ABB RobotStudio station: Proyecto_manipuladores_G3.rsstn

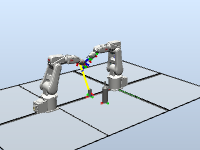
Station Proyecto_manipuladores (saved by RobotStudio format 3)
Controller Sistema8, task T_ROB1: task frame (RAPID world) sits at (1100, -1.84, 0) mm, rotated rx 0 ry 0 rz 180 deg in the station
Controller IRB_120_3kg_0.58m
  mechanical unit ROB_1: IRB120_3_58__01, 6 joints, base frame (0, 0, 0) mm
Controller Sistema8
  mechanical unit ROB_1: IRB120_3_58__01_3, 6 joints, base frame (0, 0, 0) mm
Layout (positions relative to the parent item):
  - IRB120_3_58__01 [mechanism, from Robots\IRB120_3_58_G_01.rslib] at (0, 0, 0) mm; joint values [0.0001, 0.0287, -0.0253, -0.0001, 0.5202, 0.0001] (rad or m)
  - Smart_Gripper_Servo_Fingers [mechanism, from Tools\ABB_Smart_Gripper_Servo_Fingers.rslib] at (372.35, 0.02, 592.85) mm, rotated rx 180 ry 60 rz 180 deg; joint values [0.025] (rad or m)
  - Botella_vino_objeto [part] at (0.08, -0.09, 0.03) mm, rotated rx 0 ry 0 rz 0.01 deg
  - Vaso [part] at (0, -0.1, -0.01) mm, rotated rx 0.01 ry 0 rz 0.01 deg
  - IRB120_3_58__01_3 [mechanism, from Robots\IRB120_3_58_G_01.rslib] at (1100, -1.84, 0) mm, rotated rx 0 ry 0 rz -180 deg; joint values [0, 0.3812, -0.2541, -0.0001, 0.3964, 0.0001] (rad or m)
  - Smart_Gripper_Servo_Fingers_2 [mechanism, from Tools\ABB_Smart_Gripper_Servo_Fingers.rslib] at (628.75, -1.86, 535.75) mm, rotated rx -180 ry 60 rz 0 deg; joint values [0.0221] (rad or m)
Attachment: Botella_vino is attached to Botella_vino_objeto
Attachment: Vasito is attached to Vaso
Attachment: Smart_Gripper_Servo_Fingers is attached to IRB120_3_58__01 / Link6
Attachment: Smart_Gripper_Servo_Fingers_2 is attached to IRB120_3_58__01_3 / Link6
EventTableEntry 1530: Group=, Trigger=Gripper 1531, Actions=[EventTableActionMechanicalPose 1532, EventTableActionAttach 1533], Comment=, ActivationMode=2, Cyclic=false
EventTableTriggerIO 1531: IOValue=[1], IRC5Controller=? -1, Operator=0, SignalSource=IRB_120_3kg_0.58m 521
EventTableActionMechanicalPose 1532: VirtualSignal=, Mechanism=Smart_Gripper_Servo_Fingers 1411, ToPoseName=CerradoVino, VirtualSignalValue=[1]
EventTableActionAttach 1533: AttachmentParent=Smart_Gripper_Servo_Fingers 1411, AttachmentChild=? -1, MountObject=false, Offset=[X=1, Y=0, Z=0, W=0, X=0, Y=1, Z=0, W=0, X=0, Y=0, Z=1, W=0, X=0, Y=0, Z=0, W=1], FlangeIndext=0, FindNearest=true
EventTableTriggerIO 1534: IOValue=[1], IRC5Controller=? -1, Operator=0, SignalSource=IRB_120_3kg_0.58m 521
EventTableTriggerIO 1535: IOValue=[1], IRC5Controller=? -1, Operator=0, SignalSource=IRB_120_3kg_0.58m 521
EventTableEntry 1536: Group=, Trigger=Gripper 1537, Actions=[EventTableActionMechanicalPose 1538, EventTableActionDetach 1539], Comment=, ActivationMode=2, Cyclic=false
EventTableTriggerIO 1537: IOValue=[0], IRC5Controller=? -1, Operator=0, SignalSource=IRB_120_3kg_0.58m 521
EventTableActionMechanicalPose 1538: VirtualSignal=, Mechanism=Smart_Gripper_Servo_Fingers 1411, ToPoseName=PoseAbierto, VirtualSignalValue=[1]
EventTableActionDetach 1539: AttachmentParent=Smart_Gripper_Servo_Fingers 1411, AttachmentChild=? -1
EventTableTriggerIO 1540: IOValue=[0], IRC5Controller=? -1, Operator=0, SignalSource=IRB_120_3kg_0.58m 521
EventTableTriggerIO 1541: IOValue=[0], IRC5Controller=? -1, Operator=0, SignalSource=IRB_120_3kg_0.58m 521
EventTableTriggerIO 1596: IOValue=[1], IRC5Controller=? -1, Operator=0, SignalSource=IRB_120_3kg_0.58m 521
EventTableTriggerIO 1597: IOValue=[1], IRC5Controller=? -1, Operator=0, SignalSource=IRB_120_3kg_0.58m 521
EventTableTriggerIO 1598: IOValue=[1], IRC5Controller=? -1, Operator=0, SignalSource=IRB_120_3kg_0.58m 521
EventTableTriggerIO 1599: IOValue=[0], IRC5Controller=? -1, Operator=0, SignalSource=IRB_120_3kg_0.58m 521
EventTableTriggerIO 1600: IOValue=[0], IRC5Controller=? -1, Operator=0, SignalSource=IRB_120_3kg_0.58m 521
EventTableTriggerIO 1601: IOValue=[0], IRC5Controller=? -1, Operator=0, SignalSource=IRB_120_3kg_0.58m 521
EventTableTriggerIO 1602: IOValue=[1], IRC5Controller=? -1, Operator=0, SignalSource=IRB_120_3kg_0.58m 521
EventTableTriggerIO 1603: IOValue=[0], IRC5Controller=? -1, Operator=0, SignalSource=IRB_120_3kg_0.58m 521
EventTableTriggerIO 1604: IOValue=[1], IRC5Controller=? -1, Operator=0, SignalSource=IRB_120_3kg_0.58m 521
EventTableTriggerIO 1605: IOValue=[1], IRC5Controller=? -1, Operator=0, SignalSource=IRB_120_3kg_0.58m 521
EventTableTriggerIO 1606: IOValue=[1], IRC5Controller=? -1, Operator=0, SignalSource=IRB_120_3kg_0.58m 521
EventTableTriggerIO 1607: IOValue=[1], IRC5Controller=? -1, Operator=0, SignalSource=IRB_120_3kg_0.58m 521
EventTableTriggerIO 1608: IOValue=[0], IRC5Controller=? -1, Operator=0, SignalSource=IRB_120_3kg_0.58m 521
EventTableTriggerIO 1609: IOValue=[0], IRC5Controller=? -1, Operator=0, SignalSource=IRB_120_3kg_0.58m 521
EventTableTriggerIO 1610: IOValue=[0], IRC5Controller=? -1, Operator=0, SignalSource=IRB_120_3kg_0.58m 521
EventTableTriggerIO 1611: IOValue=[0], IRC5Controller=? -1, Operator=0, SignalSource=IRB_120_3kg_0.58m 521
EventTableTriggerIO 1646: IOValue=[1], IRC5Controller=? -1, Operator=0, SignalSource=IRB_120_3kg_0.58m 521
EventTableTriggerIO 1647: IOValue=[1], IRC5Controller=? -1, Operator=0, SignalSource=IRB_120_3kg_0.58m 521
EventTableTriggerIO 1648: IOValue=[0], IRC5Controller=? -1, Operator=0, SignalSource=IRB_120_3kg_0.58m 521
EventTableTriggerIO 1649: IOValue=[0], IRC5Controller=? -1, Operator=0, SignalSource=IRB_120_3kg_0.58m 521
EventTableTriggerIO 1667: IOValue=[1], IRC5Controller=? -1, Operator=0, SignalSource=IRB_120_3kg_0.58m 521
EventTableTriggerIO 1668: IOValue=[1], IRC5Controller=? -1, Operator=0, SignalSource=IRB_120_3kg_0.58m 521
EventTableTriggerIO 1669: IOValue=[1], IRC5Controller=? -1, Operator=0, SignalSource=IRB_120_3kg_0.58m 521
EventTableTriggerIO 1670: IOValue=[1], IRC5Controller=? -1, Operator=0, SignalSource=IRB_120_3kg_0.58m 521
EventTableTriggerIO 1671: IOValue=[1], IRC5Controller=? -1, Operator=0, SignalSource=IRB_120_3kg_0.58m 521
EventTableTriggerIO 1672: IOValue=[1], IRC5Controller=? -1, Operator=0, SignalSource=IRB_120_3kg_0.58m 521
EventTableTriggerIO 1673: IOValue=[1], IRC5Controller=? -1, Operator=0, SignalSource=IRB_120_3kg_0.58m 521
EventTableTriggerIO 1674: IOValue=[1], IRC5Controller=? -1, Operator=0, SignalSource=IRB_120_3kg_0.58m 521
EventTableTriggerIO 1675: IOValue=[1], IRC5Controller=? -1, Operator=0, SignalSource=IRB_120_3kg_0.58m 521
EventTableTriggerIO 1676: IOValue=[0], IRC5Controller=? -1, Operator=0, SignalSource=IRB_120_3kg_0.58m 521
EventTableTriggerIO 1677: IOValue=[0], IRC5Controller=? -1, Operator=0, SignalSource=IRB_120_3kg_0.58m 521
EventTableTriggerIO 1678: IOValue=[0], IRC5Controller=? -1, Operator=0, SignalSource=IRB_120_3kg_0.58m 521
EventTableTriggerIO 1679: IOValue=[0], IRC5Controller=? -1, Operator=0, SignalSource=IRB_120_3kg_0.58m 521
EventTableTriggerIO 1680: IOValue=[0], IRC5Controller=? -1, Operator=0, SignalSource=IRB_120_3kg_0.58m 521
EventTableTriggerIO 1681: IOValue=[0], IRC5Controller=? -1, Operator=0, SignalSource=IRB_120_3kg_0.58m 521
EventTableTriggerIO 1682: IOValue=[0], IRC5Controller=? -1, Operator=0, SignalSource=IRB_120_3kg_0.58m 521
EventTableTriggerIO 1683: IOValue=[0], IRC5Controller=? -1, Operator=0, SignalSource=IRB_120_3kg_0.58m 521
EventTableTriggerIO 1684: IOValue=[0], IRC5Controller=? -1, Operator=0, SignalSource=IRB_120_3kg_0.58m 521
EventTableTriggerIO 2365: IOValue=[1], IRC5Controller=? -1, Operator=0, SignalSource=IRB_120_3kg_0.58m 521
EventTableTriggerIO 2366: IOValue=[1], IRC5Controller=? -1, Operator=0, SignalSource=IRB_120_3kg_0.58m 521
EventTableTriggerIO 2367: IOValue=[1], IRC5Controller=? -1, Operator=0, SignalSource=IRB_120_3kg_0.58m 521
EventTableTriggerIO 2368: IOValue=[1], IRC5Controller=? -1, Operator=0, SignalSource=IRB_120_3kg_0.58m 521
EventTableTriggerIO 2369: IOValue=[1], IRC5Controller=? -1, Operator=0, SignalSource=IRB_120_3kg_0.58m 521
EventTableTriggerIO 2370: IOValue=[1], IRC5Controller=? -1, Operator=0, SignalSource=IRB_120_3kg_0.58m 521
EventTableTriggerIO 2371: IOValue=[1], IRC5Controller=? -1, Operator=0, SignalSource=IRB_120_3kg_0.58m 521
EventTableTriggerIO 2372: IOValue=[1], IRC5Controller=? -1, Operator=0, SignalSource=IRB_120_3kg_0.58m 521
EventTableTriggerIO 2373: IOValue=[1], IRC5Controller=? -1, Operator=0, SignalSource=IRB_120_3kg_0.58m 521
EventTableTriggerIO 2374: IOValue=[0], IRC5Controller=? -1, Operator=0, SignalSource=IRB_120_3kg_0.58m 521
EventTableTriggerIO 2375: IOValue=[0], IRC5Controller=? -1, Operator=0, SignalSource=IRB_120_3kg_0.58m 521
EventTableTriggerIO 2376: IOValue=[0], IRC5Controller=? -1, Operator=0, SignalSource=IRB_120_3kg_0.58m 521
EventTableTriggerIO 2377: IOValue=[0], IRC5Controller=? -1, Operator=0, SignalSource=IRB_120_3kg_0.58m 521
EventTableTriggerIO 2378: IOValue=[0], IRC5Controller=? -1, Operator=0, SignalSource=IRB_120_3kg_0.58m 521
EventTableTriggerIO 2379: IOValue=[0], IRC5Controller=? -1, Operator=0, SignalSource=IRB_120_3kg_0.58m 521
EventTableTriggerIO 2380: IOValue=[0], IRC5Controller=? -1, Operator=0, SignalSource=IRB_120_3kg_0.58m 521
EventTableTriggerIO 2381: IOValue=[0], IRC5Controller=? -1, Operator=0, SignalSource=IRB_120_3kg_0.58m 521
EventTableTriggerIO 2382: IOValue=[0], IRC5Controller=? -1, Operator=0, SignalSource=IRB_120_3kg_0.58m 521
EventTableTriggerIO 2468: IOValue=[1], IRC5Controller=? -1, Operator=0, SignalSource=Sistema8 2502
EventTableTriggerIO 2469: IOValue=[0], IRC5Controller=? -1, Operator=0, SignalSource=Sistema8 2502
EventTableTriggerIO 2470: IOValue=[1], IRC5Controller=? -1, Operator=0, SignalSource=IRB_120_3kg_0.58m 521
EventTableTriggerIO 2471: IOValue=[1], IRC5Controller=? -1, Operator=0, SignalSource=Sistema8 2502
EventTableTriggerIO 2472: IOValue=[0], IRC5Controller=? -1, Operator=0, SignalSource=Sistema8 2502
EventTableTriggerIO 2473: IOValue=[1], IRC5Controller=? -1, Operator=0, SignalSource=IRB_120_3kg_0.58m 521
EventTableTriggerIO 2474: IOValue=[1], IRC5Controller=? -1, Operator=0, SignalSource=Sistema8 2502
EventTableTriggerIO 2475: IOValue=[0], IRC5Controller=? -1, Operator=0, SignalSource=Sistema8 2502
EventTableTriggerIO 2476: IOValue=[1], IRC5Controller=? -1, Operator=0, SignalSource=IRB_120_3kg_0.58m 521
EventTableTriggerIO 2477: IOValue=[1], IRC5Controller=? -1, Operator=0, SignalSource=Sistema8 2502
EventTableTriggerIO 2478: IOValue=[0], IRC5Controller=? -1, Operator=0, SignalSource=Sistema8 2502
EventTableTriggerIO 2479: IOValue=[1], IRC5Controller=? -1, Operator=0, SignalSource=IRB_120_3kg_0.58m 521
EventTableTriggerIO 2480: IOValue=[1], IRC5Controller=? -1, Operator=0, SignalSource=Sistema8 2502
EventTableTriggerIO 2481: IOValue=[0], IRC5Controller=? -1, Operator=0, SignalSource=Sistema8 2502
EventTableTriggerIO 2482: IOValue=[1], IRC5Controller=? -1, Operator=0, SignalSource=IRB_120_3kg_0.58m 521
EventTableTriggerIO 2483: IOValue=[1], IRC5Controller=? -1, Operator=0, SignalSource=Sistema8 2502
EventTableTriggerIO 2484: IOValue=[0], IRC5Controller=? -1, Operator=0, SignalSource=Sistema8 2502
EventTableTriggerIO 2485: IOValue=[1], IRC5Controller=? -1, Operator=0, SignalSource=IRB_120_3kg_0.58m 521
EventTableTriggerIO 2486: IOValue=[1], IRC5Controller=? -1, Operator=0, SignalSource=Sistema8 2502
EventTableTriggerIO 2487: IOValue=[0], IRC5Controller=? -1, Operator=0, SignalSource=Sistema8 2502
EventTableTriggerIO 2488: IOValue=[0], IRC5Controller=? -1, Operator=0, SignalSource=IRB_120_3kg_0.58m 521
EventTableTriggerIO 2489: IOValue=[0], IRC5Controller=? -1, Operator=0, SignalSource=IRB_120_3kg_0.58m 521
EventTableTriggerIO 2490: IOValue=[0], IRC5Controller=? -1, Operator=0, SignalSource=IRB_120_3kg_0.58m 521
EventTableTriggerIO 2491: IOValue=[0], IRC5Controller=? -1, Operator=0, SignalSource=IRB_120_3kg_0.58m 521
EventTableTriggerIO 2492: IOValue=[0], IRC5Controller=? -1, Operator=0, SignalSource=IRB_120_3kg_0.58m 521
EventTableTriggerIO 2493: IOValue=[0], IRC5Controller=? -1, Operator=0, SignalSource=IRB_120_3kg_0.58m 521
EventTableEntry 2494: Group=, Trigger=Gripper2 2468, Actions=[EventTableActionMechanicalPose 2495, EventTableActionAttach 2496], Comment=, ActivationMode=2, Cyclic=false
EventTableActionMechanicalPose 2495: VirtualSignal=, Mechanism=Smart_Gripper_Servo_Fingers_2 3134, ToPoseName=PoseAbre, VirtualSignalValue=[1]
EventTableActionAttach 2496: AttachmentParent=Smart_Gripper_Servo_Fingers_2 3134, AttachmentChild=? -1, MountObject=false, Offset=[X=1, Y=0, Z=0, W=0, X=0, Y=1, Z=0, W=0, X=0, Y=0, Z=1, W=0, X=0, Y=0, Z=0, W=1], FlangeIndext=0, FindNearest=true
EventTableEntry 2497: Group=, Trigger=Gripper2 2469, Actions=[EventTableActionMechanicalPose 3306, EventTableActionDetach 3307], Comment=, ActivationMode=2, Cyclic=false
EventTableTriggerIO 3106: IOValue=[1], IRC5Controller=? -1, Operator=0, SignalSource=IRB_120_3kg_0.58m 521
EventTableTriggerIO 3107: IOValue=[1], IRC5Controller=? -1, Operator=0, SignalSource=Sistema8 2502
EventTableTriggerIO 3108: IOValue=[0], IRC5Controller=? -1, Operator=0, SignalSource=Sistema8 2502
EventTableTriggerIO 3109: IOValue=[1], IRC5Controller=? -1, Operator=0, SignalSource=IRB_120_3kg_0.58m 521
EventTableTriggerIO 3110: IOValue=[1], IRC5Controller=? -1, Operator=0, SignalSource=Sistema8 2502
EventTableTriggerIO 3111: IOValue=[0], IRC5Controller=? -1, Operator=0, SignalSource=Sistema8 2502
EventTableTriggerIO 3112: IOValue=[1], IRC5Controller=? -1, Operator=0, SignalSource=IRB_120_3kg_0.58m 521
EventTableTriggerIO 3113: IOValue=[1], IRC5Controller=? -1, Operator=0, SignalSource=Sistema8 2502
EventTableTriggerIO 3114: IOValue=[0], IRC5Controller=? -1, Operator=0, SignalSource=Sistema8 2502
EventTableTriggerIO 3115: IOValue=[1], IRC5Controller=? -1, Operator=0, SignalSource=IRB_120_3kg_0.58m 521
EventTableTriggerIO 3116: IOValue=[1], IRC5Controller=? -1, Operator=0, SignalSource=Sistema8 2502
EventTableTriggerIO 3117: IOValue=[0], IRC5Controller=? -1, Operator=0, SignalSource=Sistema8 2502
EventTableTriggerIO 3118: IOValue=[1], IRC5Controller=? -1, Operator=0, SignalSource=IRB_120_3kg_0.58m 521
EventTableTriggerIO 3119: IOValue=[1], IRC5Controller=? -1, Operator=0, SignalSource=Sistema8 2502
EventTableTriggerIO 3120: IOValue=[0], IRC5Controller=? -1, Operator=0, SignalSource=Sistema8 2502
EventTableTriggerIO 3121: IOValue=[1], IRC5Controller=? -1, Operator=0, SignalSource=IRB_120_3kg_0.58m 521
EventTableTriggerIO 3122: IOValue=[1], IRC5Controller=? -1, Operator=0, SignalSource=Sistema8 2502
EventTableTriggerIO 3123: IOValue=[0], IRC5Controller=? -1, Operator=0, SignalSource=Sistema8 2502
EventTableTriggerIO 3124: IOValue=[0], IRC5Controller=? -1, Operator=0, SignalSource=IRB_120_3kg_0.58m 521
EventTableTriggerIO 3125: IOValue=[0], IRC5Controller=? -1, Operator=0, SignalSource=IRB_120_3kg_0.58m 521
EventTableTriggerIO 3126: IOValue=[0], IRC5Controller=? -1, Operator=0, SignalSource=IRB_120_3kg_0.58m 521
EventTableTriggerIO 3127: IOValue=[0], IRC5Controller=? -1, Operator=0, SignalSource=IRB_120_3kg_0.58m 521
EventTableTriggerIO 3128: IOValue=[0], IRC5Controller=? -1, Operator=0, SignalSource=IRB_120_3kg_0.58m 521
EventTableTriggerIO 3129: IOValue=[0], IRC5Controller=? -1, Operator=0, SignalSource=IRB_120_3kg_0.58m 521
EventTableTriggerIO 3142: IOValue=[1], IRC5Controller=? -1, Operator=0, SignalSource=IRB_120_3kg_0.58m 521
EventTableTriggerIO 3143: IOValue=[1], IRC5Controller=? -1, Operator=0, SignalSource=Sistema8 2502
EventTableTriggerIO 3144: IOValue=[0], IRC5Controller=? -1, Operator=0, SignalSource=Sistema8 2502
EventTableTriggerIO 3145: IOValue=[1], IRC5Controller=? -1, Operator=0, SignalSource=IRB_120_3kg_0.58m 521
EventTableTriggerIO 3146: IOValue=[1], IRC5Controller=? -1, Operator=0, SignalSource=Sistema8 2502
EventTableTriggerIO 3147: IOValue=[0], IRC5Controller=? -1, Operator=0, SignalSource=Sistema8 2502
EventTableTriggerIO 3148: IOValue=[1], IRC5Controller=? -1, Operator=0, SignalSource=IRB_120_3kg_0.58m 521
EventTableTriggerIO 3149: IOValue=[1], IRC5Controller=? -1, Operator=0, SignalSource=Sistema8 2502
EventTableTriggerIO 3150: IOValue=[0], IRC5Controller=? -1, Operator=0, SignalSource=Sistema8 2502
EventTableTriggerIO 3151: IOValue=[1], IRC5Controller=? -1, Operator=0, SignalSource=IRB_120_3kg_0.58m 521
EventTableTriggerIO 3152: IOValue=[1], IRC5Controller=? -1, Operator=0, SignalSource=Sistema8 2502
EventTableTriggerIO 3153: IOValue=[0], IRC5Controller=? -1, Operator=0, SignalSource=Sistema8 2502
EventTableTriggerIO 3154: IOValue=[1], IRC5Controller=? -1, Operator=0, SignalSource=IRB_120_3kg_0.58m 521
EventTableTriggerIO 3155: IOValue=[1], IRC5Controller=? -1, Operator=0, SignalSource=Sistema8 2502
EventTableTriggerIO 3156: IOValue=[0], IRC5Controller=? -1, Operator=0, SignalSource=Sistema8 2502
EventTableTriggerIO 3157: IOValue=[1], IRC5Controller=? -1, Operator=0, SignalSource=IRB_120_3kg_0.58m 521
EventTableTriggerIO 3158: IOValue=[1], IRC5Controller=? -1, Operator=0, SignalSource=Sistema8 2502
EventTableTriggerIO 3159: IOValue=[0], IRC5Controller=? -1, Operator=0, SignalSource=Sistema8 2502
EventTableTriggerIO 3160: IOValue=[1], IRC5Controller=? -1, Operator=0, SignalSource=IRB_120_3kg_0.58m 521
EventTableTriggerIO 3161: IOValue=[1], IRC5Controller=? -1, Operator=0, SignalSource=Sistema8 2502
EventTableTriggerIO 3162: IOValue=[0], IRC5Controller=? -1, Operator=0, SignalSource=Sistema8 2502
EventTableTriggerIO 3163: IOValue=[1], IRC5Controller=? -1, Operator=0, SignalSource=IRB_120_3kg_0.58m 521
EventTableTriggerIO 3164: IOValue=[1], IRC5Controller=? -1, Operator=0, SignalSource=Sistema8 2502
EventTableTriggerIO 3165: IOValue=[0], IRC5Controller=? -1, Operator=0, SignalSource=Sistema8 2502
EventTableTriggerIO 3166: IOValue=[1], IRC5Controller=? -1, Operator=0, SignalSource=IRB_120_3kg_0.58m 521
EventTableTriggerIO 3167: IOValue=[1], IRC5Controller=? -1, Operator=0, SignalSource=Sistema8 2502
EventTableTriggerIO 3168: IOValue=[0], IRC5Controller=? -1, Operator=0, SignalSource=Sistema8 2502
EventTableTriggerIO 3169: IOValue=[1], IRC5Controller=? -1, Operator=0, SignalSource=IRB_120_3kg_0.58m 521
EventTableTriggerIO 3170: IOValue=[1], IRC5Controller=? -1, Operator=0, SignalSource=Sistema8 2502
EventTableTriggerIO 3171: IOValue=[0], IRC5Controller=? -1, Operator=0, SignalSource=Sistema8 2502
EventTableTriggerIO 3172: IOValue=[1], IRC5Controller=? -1, Operator=0, SignalSource=IRB_120_3kg_0.58m 521
EventTableTriggerIO 3173: IOValue=[1], IRC5Controller=? -1, Operator=0, SignalSource=Sistema8 2502
EventTableTriggerIO 3174: IOValue=[0], IRC5Controller=? -1, Operator=0, SignalSource=Sistema8 2502
EventTableTriggerIO 3175: IOValue=[1], IRC5Controller=? -1, Operator=0, SignalSource=IRB_120_3kg_0.58m 521
EventTableTriggerIO 3176: IOValue=[1], IRC5Controller=? -1, Operator=0, SignalSource=Sistema8 2502
EventTableTriggerIO 3177: IOValue=[0], IRC5Controller=? -1, Operator=0, SignalSource=Sistema8 2502
EventTableTriggerIO 3178: IOValue=[1], IRC5Controller=? -1, Operator=0, SignalSource=IRB_120_3kg_0.58m 521
EventTableTriggerIO 3179: IOValue=[1], IRC5Controller=? -1, Operator=0, SignalSource=Sistema8 2502
EventTableTriggerIO 3180: IOValue=[0], IRC5Controller=? -1, Operator=0, SignalSource=Sistema8 2502
EventTableTriggerIO 3181: IOValue=[1], IRC5Controller=? -1, Operator=0, SignalSource=IRB_120_3kg_0.58m 521
EventTableTriggerIO 3182: IOValue=[1], IRC5Controller=? -1, Operator=0, SignalSource=Sistema8 2502
EventTableTriggerIO 3183: IOValue=[0], IRC5Controller=? -1, Operator=0, SignalSource=Sistema8 2502
EventTableTriggerIO 3184: IOValue=[1], IRC5Controller=? -1, Operator=0, SignalSource=IRB_120_3kg_0.58m 521
EventTableTriggerIO 3185: IOValue=[1], IRC5Controller=? -1, Operator=0, SignalSource=Sistema8 2502
EventTableTriggerIO 3186: IOValue=[0], IRC5Controller=? -1, Operator=0, SignalSource=Sistema8 2502
EventTableTriggerIO 3187: IOValue=[1], IRC5Controller=? -1, Operator=0, SignalSource=IRB_120_3kg_0.58m 521
EventTableTriggerIO 3188: IOValue=[1], IRC5Controller=? -1, Operator=0, SignalSource=Sistema8 2502
EventTableTriggerIO 3189: IOValue=[0], IRC5Controller=? -1, Operator=0, SignalSource=Sistema8 2502
EventTableTriggerIO 3190: IOValue=[1], IRC5Controller=? -1, Operator=0, SignalSource=IRB_120_3kg_0.58m 521
EventTableTriggerIO 3191: IOValue=[1], IRC5Controller=? -1, Operator=0, SignalSource=Sistema8 2502
EventTableTriggerIO 3192: IOValue=[0], IRC5Controller=? -1, Operator=0, SignalSource=Sistema8 2502
EventTableTriggerIO 3193: IOValue=[1], IRC5Controller=? -1, Operator=0, SignalSource=IRB_120_3kg_0.58m 521
EventTableTriggerIO 3194: IOValue=[1], IRC5Controller=? -1, Operator=0, SignalSource=Sistema8 2502
EventTableTriggerIO 3195: IOValue=[0], IRC5Controller=? -1, Operator=0, SignalSource=Sistema8 2502
EventTableTriggerIO 3196: IOValue=[1], IRC5Controller=? -1, Operator=0, SignalSource=IRB_120_3kg_0.58m 521
EventTableTriggerIO 3197: IOValue=[1], IRC5Controller=? -1, Operator=0, SignalSource=Sistema8 2502
EventTableTriggerIO 3198: IOValue=[0], IRC5Controller=? -1, Operator=0, SignalSource=Sistema8 2502
EventTableTriggerIO 3199: IOValue=[1], IRC5Controller=? -1, Operator=0, SignalSource=IRB_120_3kg_0.58m 521
EventTableTriggerIO 3200: IOValue=[1], IRC5Controller=? -1, Operator=0, SignalSource=Sistema8 2502
EventTableTriggerIO 3201: IOValue=[0], IRC5Controller=? -1, Operator=0, SignalSource=Sistema8 2502
EventTableTriggerIO 3202: IOValue=[1], IRC5Controller=? -1, Operator=0, SignalSource=IRB_120_3kg_0.58m 521
EventTableTriggerIO 3203: IOValue=[1], IRC5Controller=? -1, Operator=0, SignalSource=Sistema8 2502
EventTableTriggerIO 3204: IOValue=[0], IRC5Controller=? -1, Operator=0, SignalSource=Sistema8 2502
EventTableTriggerIO 3205: IOValue=[1], IRC5Controller=? -1, Operator=0, SignalSource=IRB_120_3kg_0.58m 521
EventTableTriggerIO 3206: IOValue=[1], IRC5Controller=? -1, Operator=0, SignalSource=Sistema8 2502
EventTableTriggerIO 3207: IOValue=[0], IRC5Controller=? -1, Operator=0, SignalSource=Sistema8 2502
EventTableTriggerIO 3208: IOValue=[1], IRC5Controller=? -1, Operator=0, SignalSource=IRB_120_3kg_0.58m 521
EventTableTriggerIO 3209: IOValue=[1], IRC5Controller=? -1, Operator=0, SignalSource=Sistema8 2502
EventTableTriggerIO 3210: IOValue=[0], IRC5Controller=? -1, Operator=0, SignalSource=Sistema8 2502
EventTableTriggerIO 3211: IOValue=[1], IRC5Controller=? -1, Operator=0, SignalSource=IRB_120_3kg_0.58m 521
EventTableTriggerIO 3212: IOValue=[1], IRC5Controller=? -1, Operator=0, SignalSource=Sistema8 2502
EventTableTriggerIO 3213: IOValue=[0], IRC5Controller=? -1, Operator=0, SignalSource=Sistema8 2502
EventTableTriggerIO 3214: IOValue=[1], IRC5Controller=? -1, Operator=0, SignalSource=IRB_120_3kg_0.58m 521
EventTableTriggerIO 3215: IOValue=[1], IRC5Controller=? -1, Operator=0, SignalSource=Sistema8 2502
EventTableTriggerIO 3216: IOValue=[0], IRC5Controller=? -1, Operator=0, SignalSource=Sistema8 2502
EventTableTriggerIO 3217: IOValue=[1], IRC5Controller=? -1, Operator=0, SignalSource=IRB_120_3kg_0.58m 521
EventTableTriggerIO 3218: IOValue=[1], IRC5Controller=? -1, Operator=0, SignalSource=Sistema8 2502
EventTableTriggerIO 3219: IOValue=[0], IRC5Controller=? -1, Operator=0, SignalSource=Sistema8 2502
EventTableTriggerIO 3220: IOValue=[1], IRC5Controller=? -1, Operator=0, SignalSource=IRB_120_3kg_0.58m 521
EventTableTriggerIO 3221: IOValue=[1], IRC5Controller=? -1, Operator=0, SignalSource=Sistema8 2502
EventTableTriggerIO 3222: IOValue=[0], IRC5Controller=? -1, Operator=0, SignalSource=Sistema8 2502
EventTableTriggerIO 3223: IOValue=[1], IRC5Controller=? -1, Operator=0, SignalSource=IRB_120_3kg_0.58m 521
EventTableTriggerIO 3224: IOValue=[1], IRC5Controller=? -1, Operator=0, SignalSource=Sistema8 2502
EventTableTriggerIO 3225: IOValue=[0], IRC5Controller=? -1, Operator=0, SignalSource=Sistema8 2502
EventTableTriggerIO 3226: IOValue=[1], IRC5Controller=? -1, Operator=0, SignalSource=IRB_120_3kg_0.58m 521
EventTableTriggerIO 3227: IOValue=[1], IRC5Controller=? -1, Operator=0, SignalSource=Sistema8 2502
EventTableTriggerIO 3228: IOValue=[0], IRC5Controller=? -1, Operator=0, SignalSource=Sistema8 2502
EventTableTriggerIO 3229: IOValue=[1], IRC5Controller=? -1, Operator=0, SignalSource=IRB_120_3kg_0.58m 521
EventTableTriggerIO 3230: IOValue=[1], IRC5Controller=? -1, Operator=0, SignalSource=Sistema8 2502
EventTableTriggerIO 3231: IOValue=[0], IRC5Controller=? -1, Operator=0, SignalSource=Sistema8 2502
EventTableTriggerIO 3232: IOValue=[1], IRC5Controller=? -1, Operator=0, SignalSource=IRB_120_3kg_0.58m 521
EventTableTriggerIO 3233: IOValue=[1], IRC5Controller=? -1, Operator=0, SignalSource=Sistema8 2502
EventTableTriggerIO 3234: IOValue=[0], IRC5Controller=? -1, Operator=0, SignalSource=Sistema8 2502
EventTableTriggerIO 3235: IOValue=[1], IRC5Controller=? -1, Operator=0, SignalSource=IRB_120_3kg_0.58m 521
EventTableTriggerIO 3236: IOValue=[1], IRC5Controller=? -1, Operator=0, SignalSource=Sistema8 2502
EventTableTriggerIO 3237: IOValue=[0], IRC5Controller=? -1, Operator=0, SignalSource=Sistema8 2502
EventTableTriggerIO 3238: IOValue=[1], IRC5Controller=? -1, Operator=0, SignalSource=IRB_120_3kg_0.58m 521
EventTableTriggerIO 3239: IOValue=[1], IRC5Controller=? -1, Operator=0, SignalSource=Sistema8 2502
EventTableTriggerIO 3240: IOValue=[0], IRC5Controller=? -1, Operator=0, SignalSource=Sistema8 2502
EventTableTriggerIO 3241: IOValue=[1], IRC5Controller=? -1, Operator=0, SignalSource=IRB_120_3kg_0.58m 521
EventTableTriggerIO 3242: IOValue=[1], IRC5Controller=? -1, Operator=0, SignalSource=Sistema8 2502
EventTableTriggerIO 3243: IOValue=[0], IRC5Controller=? -1, Operator=0, SignalSource=Sistema8 2502
EventTableTriggerIO 3244: IOValue=[1], IRC5Controller=? -1, Operator=0, SignalSource=IRB_120_3kg_0.58m 521
EventTableTriggerIO 3245: IOValue=[1], IRC5Controller=? -1, Operator=0, SignalSource=Sistema8 2502
EventTableTriggerIO 3246: IOValue=[0], IRC5Controller=? -1, Operator=0, SignalSource=Sistema8 2502
EventTableTriggerIO 3247: IOValue=[1], IRC5Controller=? -1, Operator=0, SignalSource=IRB_120_3kg_0.58m 521
EventTableTriggerIO 3248: IOValue=[1], IRC5Controller=? -1, Operator=0, SignalSource=Sistema8 2502
EventTableTriggerIO 3249: IOValue=[0], IRC5Controller=? -1, Operator=0, SignalSource=Sistema8 2502
EventTableTriggerIO 3250: IOValue=[1], IRC5Controller=? -1, Operator=0, SignalSource=IRB_120_3kg_0.58m 521
EventTableTriggerIO 3251: IOValue=[1], IRC5Controller=? -1, Operator=0, SignalSource=Sistema8 2502
EventTableTriggerIO 3252: IOValue=[0], IRC5Controller=? -1, Operator=0, SignalSource=Sistema8 2502
EventTableTriggerIO 3253: IOValue=[1], IRC5Controller=? -1, Operator=0, SignalSource=IRB_120_3kg_0.58m 521
EventTableTriggerIO 3254: IOValue=[1], IRC5Controller=? -1, Operator=0, SignalSource=Sistema8 2502
EventTableTriggerIO 3255: IOValue=[0], IRC5Controller=? -1, Operator=0, SignalSource=Sistema8 2502
EventTableTriggerIO 3256: IOValue=[1], IRC5Controller=? -1, Operator=0, SignalSource=IRB_120_3kg_0.58m 521
EventTableTriggerIO 3257: IOValue=[1], IRC5Controller=? -1, Operator=0, SignalSource=Sistema8 2502
EventTableTriggerIO 3258: IOValue=[0], IRC5Controller=? -1, Operator=0, SignalSource=Sistema8 2502
EventTableTriggerIO 3259: IOValue=[1], IRC5Controller=? -1, Operator=0, SignalSource=IRB_120_3kg_0.58m 521
EventTableTriggerIO 3260: IOValue=[1], IRC5Controller=? -1, Operator=0, SignalSource=Sistema8 2502
EventTableTriggerIO 3261: IOValue=[0], IRC5Controller=? -1, Operator=0, SignalSource=Sistema8 2502
EventTableTriggerIO 3262: IOValue=[1], IRC5Controller=? -1, Operator=0, SignalSource=IRB_120_3kg_0.58m 521
EventTableTriggerIO 3263: IOValue=[1], IRC5Controller=? -1, Operator=0, SignalSource=Sistema8 2502
EventTableTriggerIO 3264: IOValue=[0], IRC5Controller=? -1, Operator=0, SignalSource=Sistema8 2502
EventTableTriggerIO 3265: IOValue=[0], IRC5Controller=? -1, Operator=0, SignalSource=IRB_120_3kg_0.58m 521
EventTableTriggerIO 3266: IOValue=[0], IRC5Controller=? -1, Operator=0, SignalSource=IRB_120_3kg_0.58m 521
EventTableTriggerIO 3267: IOValue=[0], IRC5Controller=? -1, Operator=0, SignalSource=IRB_120_3kg_0.58m 521
EventTableTriggerIO 3268: IOValue=[0], IRC5Controller=? -1, Operator=0, SignalSource=IRB_120_3kg_0.58m 521
EventTableTriggerIO 3269: IOValue=[0], IRC5Controller=? -1, Operator=0, SignalSource=IRB_120_3kg_0.58m 521
EventTableTriggerIO 3270: IOValue=[0], IRC5Controller=? -1, Operator=0, SignalSource=IRB_120_3kg_0.58m 521
EventTableTriggerIO 3271: IOValue=[0], IRC5Controller=? -1, Operator=0, SignalSource=IRB_120_3kg_0.58m 521
EventTableTriggerIO 3272: IOValue=[0], IRC5Controller=? -1, Operator=0, SignalSource=IRB_120_3kg_0.58m 521
EventTableTriggerIO 3273: IOValue=[0], IRC5Controller=? -1, Operator=0, SignalSource=IRB_120_3kg_0.58m 521
EventTableTriggerIO 3274: IOValue=[0], IRC5Controller=? -1, Operator=0, SignalSource=IRB_120_3kg_0.58m 521
EventTableTriggerIO 3275: IOValue=[0], IRC5Controller=? -1, Operator=0, SignalSource=IRB_120_3kg_0.58m 521
EventTableTriggerIO 3276: IOValue=[0], IRC5Controller=? -1, Operator=0, SignalSource=IRB_120_3kg_0.58m 521
EventTableTriggerIO 3277: IOValue=[0], IRC5Controller=? -1, Operator=0, SignalSource=IRB_120_3kg_0.58m 521
EventTableTriggerIO 3278: IOValue=[0], IRC5Controller=? -1, Operator=0, SignalSource=IRB_120_3kg_0.58m 521
EventTableTriggerIO 3279: IOValue=[0], IRC5Controller=? -1, Operator=0, SignalSource=IRB_120_3kg_0.58m 521
EventTableTriggerIO 3280: IOValue=[0], IRC5Controller=? -1, Operator=0, SignalSource=IRB_120_3kg_0.58m 521
EventTableTriggerIO 3281: IOValue=[0], IRC5Controller=? -1, Operator=0, SignalSource=IRB_120_3kg_0.58m 521
EventTableTriggerIO 3282: IOValue=[0], IRC5Controller=? -1, Operator=0, SignalSource=IRB_120_3kg_0.58m 521
EventTableTriggerIO 3283: IOValue=[0], IRC5Controller=? -1, Operator=0, SignalSource=IRB_120_3kg_0.58m 521
EventTableTriggerIO 3284: IOValue=[0], IRC5Controller=? -1, Operator=0, SignalSource=IRB_120_3kg_0.58m 521
EventTableTriggerIO 3285: IOValue=[0], IRC5Controller=? -1, Operator=0, SignalSource=IRB_120_3kg_0.58m 521
EventTableTriggerIO 3286: IOValue=[0], IRC5Controller=? -1, Operator=0, SignalSource=IRB_120_3kg_0.58m 521
EventTableTriggerIO 3287: IOValue=[0], IRC5Controller=? -1, Operator=0, SignalSource=IRB_120_3kg_0.58m 521
EventTableTriggerIO 3288: IOValue=[0], IRC5Controller=? -1, Operator=0, SignalSource=IRB_120_3kg_0.58m 521
EventTableTriggerIO 3289: IOValue=[0], IRC5Controller=? -1, Operator=0, SignalSource=IRB_120_3kg_0.58m 521
EventTableTriggerIO 3290: IOValue=[0], IRC5Controller=? -1, Operator=0, SignalSource=IRB_120_3kg_0.58m 521
EventTableTriggerIO 3291: IOValue=[0], IRC5Controller=? -1, Operator=0, SignalSource=IRB_120_3kg_0.58m 521
EventTableTriggerIO 3292: IOValue=[0], IRC5Controller=? -1, Operator=0, SignalSource=IRB_120_3kg_0.58m 521
EventTableTriggerIO 3293: IOValue=[0], IRC5Controller=? -1, Operator=0, SignalSource=IRB_120_3kg_0.58m 521
EventTableTriggerIO 3294: IOValue=[0], IRC5Controller=? -1, Operator=0, SignalSource=IRB_120_3kg_0.58m 521
EventTableTriggerIO 3295: IOValue=[0], IRC5Controller=? -1, Operator=0, SignalSource=IRB_120_3kg_0.58m 521
EventTableTriggerIO 3296: IOValue=[0], IRC5Controller=? -1, Operator=0, SignalSource=IRB_120_3kg_0.58m 521
EventTableTriggerIO 3297: IOValue=[0], IRC5Controller=? -1, Operator=0, SignalSource=IRB_120_3kg_0.58m 521
EventTableTriggerIO 3298: IOValue=[0], IRC5Controller=? -1, Operator=0, SignalSource=IRB_120_3kg_0.58m 521
EventTableTriggerIO 3299: IOValue=[0], IRC5Controller=? -1, Operator=0, SignalSource=IRB_120_3kg_0.58m 521
EventTableTriggerIO 3300: IOValue=[0], IRC5Controller=? -1, Operator=0, SignalSource=IRB_120_3kg_0.58m 521
EventTableTriggerIO 3301: IOValue=[0], IRC5Controller=? -1, Operator=0, SignalSource=IRB_120_3kg_0.58m 521
EventTableTriggerIO 3302: IOValue=[0], IRC5Controller=? -1, Operator=0, SignalSource=IRB_120_3kg_0.58m 521
EventTableTriggerIO 3303: IOValue=[0], IRC5Controller=? -1, Operator=0, SignalSource=IRB_120_3kg_0.58m 521
EventTableTriggerIO 3304: IOValue=[0], IRC5Controller=? -1, Operator=0, SignalSource=IRB_120_3kg_0.58m 521
EventTableTriggerIO 3305: IOValue=[0], IRC5Controller=? -1, Operator=0, SignalSource=IRB_120_3kg_0.58m 521
EventTableActionMechanicalPose 3306: VirtualSignal=, Mechanism=Smart_Gripper_Servo_Fingers_2 3134, ToPoseName=PoseCerrado, VirtualSignalValue=[1]
EventTableActionDetach 3307: AttachmentParent=Smart_Gripper_Servo_Fingers_2 3134, AttachmentChild=? -1
EventTableTriggerIO 3389: IOValue=[1], IRC5Controller=? -1, Operator=0, SignalSource=IRB_120_3kg_0.58m 521
EventTableTriggerIO 3390: IOValue=[1], IRC5Controller=? -1, Operator=0, SignalSource=Sistema8 2502
EventTableTriggerIO 3391: IOValue=[0], IRC5Controller=? -1, Operator=0, SignalSource=Sistema8 2502
EventTableTriggerIO 3392: IOValue=[1], IRC5Controller=? -1, Operator=0, SignalSource=IRB_120_3kg_0.58m 521
EventTableTriggerIO 3393: IOValue=[1], IRC5Controller=? -1, Operator=0, SignalSource=Sistema8 2502
EventTableTriggerIO 3394: IOValue=[0], IRC5Controller=? -1, Operator=0, SignalSource=Sistema8 2502
EventTableTriggerIO 3395: IOValue=[1], IRC5Controller=? -1, Operator=0, SignalSource=IRB_120_3kg_0.58m 521
EventTableTriggerIO 3396: IOValue=[1], IRC5Controller=? -1, Operator=0, SignalSource=Sistema8 2502
EventTableTriggerIO 3397: IOValue=[0], IRC5Controller=? -1, Operator=0, SignalSource=Sistema8 2502
EventTableTriggerIO 3398: IOValue=[1], IRC5Controller=? -1, Operator=0, SignalSource=IRB_120_3kg_0.58m 521
EventTableTriggerIO 3399: IOValue=[1], IRC5Controller=? -1, Operator=0, SignalSource=Sistema8 2502
EventTableTriggerIO 3400: IOValue=[0], IRC5Controller=? -1, Operator=0, SignalSource=Sistema8 2502
EventTableTriggerIO 3401: IOValue=[1], IRC5Controller=? -1, Operator=0, SignalSource=IRB_120_3kg_0.58m 521
EventTableTriggerIO 3402: IOValue=[1], IRC5Controller=? -1, Operator=0, SignalSource=Sistema8 2502
EventTableTriggerIO 3403: IOValue=[0], IRC5Controller=? -1, Operator=0, SignalSource=Sistema8 2502
EventTableTriggerIO 3404: IOValue=[1], IRC5Controller=? -1, Operator=0, SignalSource=IRB_120_3kg_0.58m 521
EventTableTriggerIO 3405: IOValue=[1], IRC5Controller=? -1, Operator=0, SignalSource=Sistema8 2502
EventTableTriggerIO 3406: IOValue=[0], IRC5Controller=? -1, Operator=0, SignalSource=Sistema8 2502
EventTableTriggerIO 3407: IOValue=[1], IRC5Controller=? -1, Operator=0, SignalSource=IRB_120_3kg_0.58m 521
EventTableTriggerIO 3408: IOValue=[1], IRC5Controller=? -1, Operator=0, SignalSource=Sistema8 2502
EventTableTriggerIO 3409: IOValue=[0], IRC5Controller=? -1, Operator=0, SignalSource=Sistema8 2502
EventTableTriggerIO 3410: IOValue=[1], IRC5Controller=? -1, Operator=0, SignalSource=IRB_120_3kg_0.58m 521
EventTableTriggerIO 3411: IOValue=[1], IRC5Controller=? -1, Operator=0, SignalSource=Sistema8 2502
EventTableTriggerIO 3412: IOValue=[0], IRC5Controller=? -1, Operator=0, SignalSource=Sistema8 2502
EventTableTriggerIO 3413: IOValue=[1], IRC5Controller=? -1, Operator=0, SignalSource=IRB_120_3kg_0.58m 521
EventTableTriggerIO 3414: IOValue=[1], IRC5Controller=? -1, Operator=0, SignalSource=Sistema8 2502
EventTableTriggerIO 3415: IOValue=[0], IRC5Controller=? -1, Operator=0, SignalSource=Sistema8 2502
EventTableTriggerIO 3416: IOValue=[1], IRC5Controller=? -1, Operator=0, SignalSource=IRB_120_3kg_0.58m 521
EventTableTriggerIO 3417: IOValue=[1], IRC5Controller=? -1, Operator=0, SignalSource=Sistema8 2502
EventTableTriggerIO 3418: IOValue=[0], IRC5Controller=? -1, Operator=0, SignalSource=Sistema8 2502
EventTableTriggerIO 3419: IOValue=[1], IRC5Controller=? -1, Operator=0, SignalSource=IRB_120_3kg_0.58m 521
EventTableTriggerIO 3420: IOValue=[1], IRC5Controller=? -1, Operator=0, SignalSource=Sistema8 2502
EventTableTriggerIO 3421: IOValue=[0], IRC5Controller=? -1, Operator=0, SignalSource=Sistema8 2502
EventTableTriggerIO 3422: IOValue=[1], IRC5Controller=? -1, Operator=0, SignalSource=IRB_120_3kg_0.58m 521
EventTableTriggerIO 3423: IOValue=[1], IRC5Controller=? -1, Operator=0, SignalSource=Sistema8 2502
EventTableTriggerIO 3424: IOValue=[0], IRC5Controller=? -1, Operator=0, SignalSource=Sistema8 2502
EventTableTriggerIO 3425: IOValue=[1], IRC5Controller=? -1, Operator=0, SignalSource=IRB_120_3kg_0.58m 521
EventTableTriggerIO 3426: IOValue=[1], IRC5Controller=? -1, Operator=0, SignalSource=Sistema8 2502
EventTableTriggerIO 3427: IOValue=[0], IRC5Controller=? -1, Operator=0, SignalSource=Sistema8 2502
EventTableTriggerIO 3428: IOValue=[1], IRC5Controller=? -1, Operator=0, SignalSource=IRB_120_3kg_0.58m 521
EventTableTriggerIO 3429: IOValue=[1], IRC5Controller=? -1, Operator=0, SignalSource=Sistema8 2502
EventTableTriggerIO 3430: IOValue=[0], IRC5Controller=? -1, Operator=0, SignalSource=Sistema8 2502
EventTableTriggerIO 3431: IOValue=[1], IRC5Controller=? -1, Operator=0, SignalSource=IRB_120_3kg_0.58m 521
EventTableTriggerIO 3432: IOValue=[1], IRC5Controller=? -1, Operator=0, SignalSource=Sistema8 2502
EventTableTriggerIO 3433: IOValue=[0], IRC5Controller=? -1, Operator=0, SignalSource=Sistema8 2502
EventTableTriggerIO 3434: IOValue=[1], IRC5Controller=? -1, Operator=0, SignalSource=IRB_120_3kg_0.58m 521
EventTableTriggerIO 3435: IOValue=[1], IRC5Controller=? -1, Operator=0, SignalSource=Sistema8 2502
EventTableTriggerIO 3436: IOValue=[0], IRC5Controller=? -1, Operator=0, SignalSource=Sistema8 2502
EventTableTriggerIO 3437: IOValue=[0], IRC5Controller=? -1, Operator=0, SignalSource=IRB_120_3kg_0.58m 521
EventTableTriggerIO 3438: IOValue=[0], IRC5Controller=? -1, Operator=0, SignalSource=IRB_120_3kg_0.58m 521
EventTableTriggerIO 3439: IOValue=[0], IRC5Controller=? -1, Operator=0, SignalSource=IRB_120_3kg_0.58m 521
EventTableTriggerIO 3440: IOValue=[0], IRC5Controller=? -1, Operator=0, SignalSource=IRB_120_3kg_0.58m 521
EventTableTriggerIO 3441: IOValue=[0], IRC5Controller=? -1, Operator=0, SignalSource=IRB_120_3kg_0.58m 521
EventTableTriggerIO 3442: IOValue=[0], IRC5Controller=? -1, Operator=0, SignalSource=IRB_120_3kg_0.58m 521
EventTableTriggerIO 3443: IOValue=[0], IRC5Controller=? -1, Operator=0, SignalSource=IRB_120_3kg_0.58m 521
EventTableTriggerIO 3444: IOValue=[0], IRC5Controller=? -1, Operator=0, SignalSource=IRB_120_3kg_0.58m 521
EventTableTriggerIO 3445: IOValue=[0], IRC5Controller=? -1, Operator=0, SignalSource=IRB_120_3kg_0.58m 521
EventTableTriggerIO 3446: IOValue=[0], IRC5Controller=? -1, Operator=0, SignalSource=IRB_120_3kg_0.58m 521
EventTableTriggerIO 3447: IOValue=[0], IRC5Controller=? -1, Operator=0, SignalSource=IRB_120_3kg_0.58m 521
EventTableTriggerIO 3448: IOValue=[0], IRC5Controller=? -1, Operator=0, SignalSource=IRB_120_3kg_0.58m 521
EventTableTriggerIO 3449: IOValue=[0], IRC5Controller=? -1, Operator=0, SignalSource=IRB_120_3kg_0.58m 521
EventTableTriggerIO 3450: IOValue=[0], IRC5Controller=? -1, Operator=0, SignalSource=IRB_120_3kg_0.58m 521
EventTableTriggerIO 3451: IOValue=[0], IRC5Controller=? -1, Operator=0, SignalSource=IRB_120_3kg_0.58m 521
EventTableTriggerIO 3452: IOValue=[0], IRC5Controller=? -1, Operator=0, SignalSource=IRB_120_3kg_0.58m 521
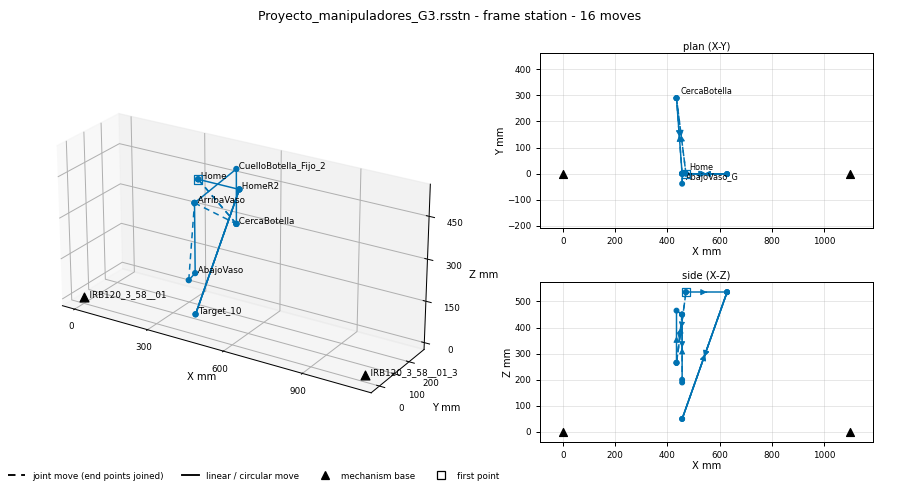
[picture p0: tool path of Proyecto_manipuladores_G3.rsstn in frame station, 16 of 16 moves have a stored position in this frame; points joined in program order, loops and branches not executed]
Targets, tools, work objects and paths stored in the station, written as RAPID:
! task T_ROB1
MODULE CalibData
  PERS tooldata MyTool:=[TRUE,[[31.792631019,0,229.638935148],[0.945518576,0,0.325568154,0]],[1,[0,0,1],[1,0,0,0],0,0,0]];
  TASK PERS wobjdata Botella_vino:=[FALSE,TRUE,"",[[435.10948997,289.246438052,0.058654266],[0.999999998,-0.000005202,-0.000035595,0.000056146]],[[0,0,0],[1,0,0,0]]];
  TASK PERS wobjdata Vasito:=[FALSE,TRUE,"",[[456.611678196,-0.00254491,0.029267825],[0.999999988,0.00010633,-0.000042508,0.000103336]],[[0,0,0],[1,0,0,0]]];
  PERS tooldata Tooldata_5:=[TRUE,[[0,0,114.2],[1,0,0,0]],[0.215,[8.7,12.3,49.2],[1,0,0,0],0.00021,0.00024,0.00009]];
  PERS tooldata Servo:=[TRUE,[[0,0,114.2],[1,0,0,0]],[0.215,[8.7,12.3,49.2],[1,0,0,0],0.00021,0.00024,0.00009]];
ENDMODULE

! task T_ROB1
MODULE Module1
  CONST robtarget Target_1:=[[349.573039208,-298.211835697,349.916285054],[0.000007053,0.707477651,-0.706735707,0.000117681],[0,0,0,0],[9E9,9E9,9E9,9E9,9E9,9E9]];
  CONST robtarget Home:=[[471.249,0.018,535.748],[0.5,0,0.866025404,0],[0,0,0,0],[9E9,9E9,9E9,9E9,9E9,9E9]];
  CONST robtarget Target_0:=[[349.560515676,-298.197730224,429.91628283],[0.000007053,0.707477651,-0.706735707,0.000117681],[0,0,0,0],[9E9,9E9,9E9,9E9,9E9,9E9]];
  CONST robtarget Soltar:=[[349.592,-298.228,350.04],[0.000007053,0.707477648,-0.706735709,0.000117666],[0,0,0,0],[9E9,9E9,9E9,9E9,9E9,9E9]];
  CONST robtarget CuelloBotella:=[[-0.000025258,-0.000123304,264.999964739],[0.707106717,-0.707106845,-0.0000002,-0.000000292],[0,1,1,0],[9E9,9E9,9E9,9E9,9E9,9E9]];
  CONST robtarget CercaBotella:=[[-0.000025258,-0.000123304,264.999964739],[0.707106717,-0.707106845,-0.0000002,-0.000000292],[0,1,1,0],[9E9,9E9,9E9,9E9,9E9,9E9]];
  CONST robtarget CuelloBotella_Fijo:=[[435.063,289.291,265],[0.707106781,-0.707106781,0,0],[0,0,0,0],[9E9,9E9,9E9,9E9,9E9,9E9]];
  CONST robtarget ArribaVaso:=[[-0.057940584,0.027004038,449.999986379],[0.707043111,-0.707170419,-0.000161782,-0.000111348],[0,0,0,0],[9E9,9E9,9E9,9E9,9E9,9E9]];
  CONST robtarget CuelloBotella_Fijo_2:=[[435.063,289.291,465],[0.707106781,-0.707106781,0,0],[0,0,0,0],[9E9,9E9,9E9,9E9,9E9,9E9]];
  CONST robtarget AbajoVaso:=[[0.038627056,-0.018002692,200.000009081],[0.382600256,-0.92391396,-0.000106857,-0.000164783],[0,0,0,0],[9E9,9E9,9E9,9E9,9E9,9E9]];
  CONST robtarget ArribaVasoG:=[[-0.057940584,0.027004038,449.999986379],[0.382600256,-0.92391396,-0.000106857,-0.000164783],[0,0,0,0],[9E9,9E9,9E9,9E9,9E9,9E9]];
  CONST robtarget AbajoVaso_G:=[[0.045380531,-38.656898793,189.654204982],[0.130436939,-0.991456588,-0.000060567,-0.000186825],[0,0,0,0],[9E9,9E9,9E9,9E9,9E9,9E9]];
  PROC Path_10()
    MoveJ Home,v1000,fine,Servo\WObj:=wobj0;
    MoveJ CercaBotella,v1000,fine,Servo\WObj:=Botella_vino;
    Reset Gripper;
    MoveJ CuelloBotella,v1000,fine,Servo\WObj:=Botella_vino;
    Set Gripper;
    MoveL CuelloBotella_Fijo_2,v1000,fine,Servo\WObj:=wobj0;
    MoveL ArribaVaso,v1000,fine,Servo\WObj:=Vasito;
    MoveJ ArribaVasoG,v1000,fine,Servo\WObj:=Vasito;
    MoveL AbajoVaso,v1000,fine,Servo\WObj:=Vasito;
    MoveL AbajoVaso_G,v1000,fine,Servo\WObj:=Vasito;
    WaitTime 3;
    MoveJ ArribaVasoG,v1000,fine,Servo\WObj:=Vasito;
    MoveJ CuelloBotella_Fijo,v1000,fine,Servo\WObj:=wobj0;
    Reset Gripper;
    MoveJ Home,v1000,fine,Servo\WObj:=wobj0;
  ENDPROC
ENDMODULE

! task T_ROB1
MODULE CalibData
  TASK PERS wobjdata Vasito:=[FALSE,TRUE,"",[[643.359080892,-1.8275672,0.123425138],[1,0.000002283,0.000002677,-0.00000561]],[[0,0,0],[1,0,0,0]]];
  PERS tooldata Servo1:=[TRUE,[[0,0,114.2],[1,0,0,0]],[0.215,[8.7,12.3,49.2],[1,0,0,0],0.00021,0.00024,0.00009]];
  PERS tooldata Servo2:=[TRUE,[[0,0,114.2],[1,0,0,0]],[0.215,[8.7,12.3,49.2],[1,0,0,0],0.00021,0.00024,0.00009]];
  PERS tooldata Servo:=[TRUE,[[0,0,114.2],[1,0,0,0]],[0.215,[8.7,12.3,49.2],[1,0,0,0],0.00021,0.00024,0.00009]];
ENDMODULE

! task T_ROB1
MODULE Module1
  CONST robtarget HomeR2:=[[471.249,0.018,535.748],[0.500000338,0.000000147,0.866025209,0.000000103],[0,0,0,0],[9E9,9E9,9E9,9E9,9E9,9E9]];
  CONST robtarget Target_10:=[[0.000347928,0.000205066,49.876574862],[0.18301346,-0.683016605,0.683009778,-0.183008288],[0,0,0,0],[9E9,9E9,9E9,9E9,9E9,9E9]];
  CONST robtarget Inter:=[[471.249,0.018,535.748],[0.500000338,0.000000147,0.866025209,0.000000103],[0,0,0,0],[9E9,9E9,9E9,9E9,9E9,9E9]];
  PROC Path_10()
    MoveL HomeR2,v1000,fine,Servo\WObj:=wobj0;
    MoveL Target_10,v1000,fine,Servo\WObj:=Vasito;
    Set Gripper2;
    MoveL Inter,v1000,fine,Servo\WObj:=wobj0;
    WaitTime 3;
    MoveL Target_10,v1000,fine,Servo\WObj:=Vasito;
    Reset Gripper2;
    MoveJ HomeR2,v1000,z100,tool0\WObj:=wobj0;
  ENDPROC
ENDMODULE

